TYPE E_LIGHTSTATE :
(
	Off,
	BlinkSlow,
	BlinkFast,
	On
);
END_TYPE

(* stored: Version 1.1.0.1, ProductVersion 3.1.0.36
   DUT E_LIGHTSTATE: Id {be89386a-9bcb-48a0-ac2c-45ae69d612ed} *)
